FUNCTION_BLOCK FeedOCSLB (* CAT Function Block Type *)
  (* Standard: 61499-2 *)
  (* Version 0.0, 6/7/2026, Schneider Electric, template *)
  PACKAGE SE.Nereda;
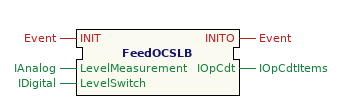
  EVENT_INPUT
    INIT;
  END_EVENT
  EVENT_OUTPUT
    INITO;
  END_EVENT
  SOCKETS
    LevelMeasurement : IAnalog;
    LevelSwitch : IDigital;
  END_SOCKETS
  PLUGS
    IOpCdt : IOpCdtItems;
  END_PLUGS
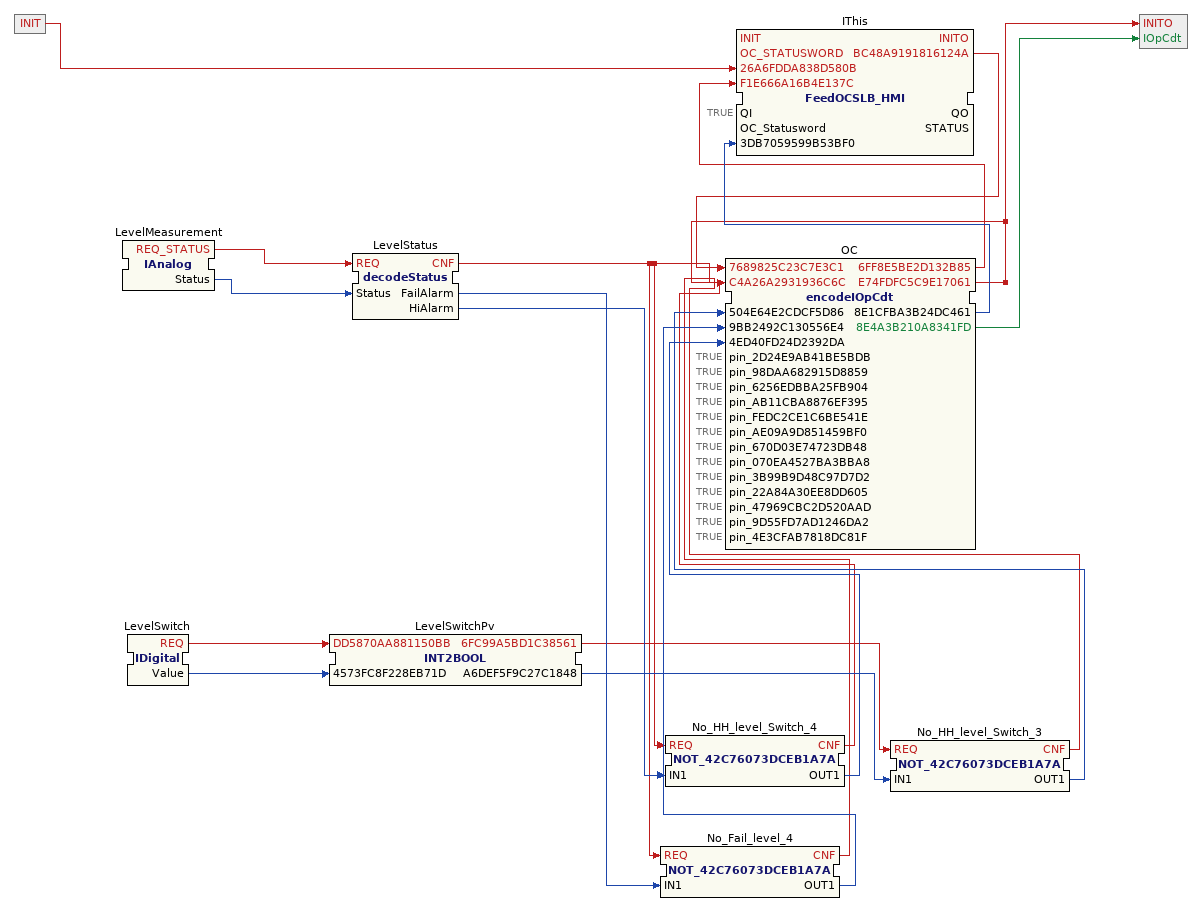
  (* 01 - FUNCTIONNAL INPUT INTERFACE *)
  (* 00 - INITIALIZATION *)
  (* 05 - LOGIC *)
  (* 06 - HMI INTERFACE *)
  (* 03 - FIELD INTERFACE *)
  (* 02 - FUNCTIONNAL OUTPUT INTERFACE *)
  (* Operating Condition Status *)
  (* Operating conditions : 1. Reserved, do not use. 2. No High level in the sludge buffer 49LT0001 3. HighHigh level switch 49LS0002 not activated 4. Level measurement 49LT0001 available *)
  FBS
    OC : encodeIOpCdt(pin_2D24E9AB41BE5BDB := TRUE, pin_98DAA682915D8859 := TRUE, pin_6256EDBBA25FB904 := TRUE, pin_AB11CBA8876EF395 := TRUE, pin_FEDC2CE1C6BE541E := TRUE, pin_AE09A9D851459BF0 := TRUE, pin_670D03E74723DB48 := TRUE, pin_070EA4527BA3BBA8 := TRUE, pin_3B99B9D48C97D7D2 := TRUE, pin_22A84A30EE8DD605 := TRUE, pin_47969CBC2D520AAD := TRUE, pin_9D55FD7AD1246DA2 := TRUE, pin_4E3CFAB7818DC81F := TRUE); (* You set the operating conditions. For the inputs that are not used set a constant to TRUE. *)
    IThis : FeedOCSLB_HMI(QI := TRUE);
    No_HH_level_Switch_3 : NOT_42C76073DCEB1A7A; {SET_ATTRIBUTE(Configuration.GenericFBType.InterfaceParams, Runtime.Standard#CNT:=1;OUT${CNT$}:BOOL)}
    LevelStatus : decodeStatus; {SET_ATTRIBUTE(Configuration.Component.HideUnusedPorts, )}
    LevelSwitchPv : INT2BOOL;
    No_Fail_level_4 : NOT_42C76073DCEB1A7A; {SET_ATTRIBUTE(Configuration.GenericFBType.InterfaceParams, Runtime.Standard#CNT:=1;OUT${CNT$}:BOOL)}
    No_HH_level_Switch_4 : NOT_42C76073DCEB1A7A; {SET_ATTRIBUTE(Configuration.GenericFBType.InterfaceParams, Runtime.Standard#CNT:=1;OUT${CNT$}:BOOL)}
  END_FBS
  EVENT_CONNECTIONS
    INIT TO IThis.26A6FDDA838D580B;
    OC.6FF8E5BE2D132B85 TO IThis.F1E666A16B4E137C;
    IThis.BC48A9191816124A TO OC.7689825C23C7E3C1;
    OC.E74FDFC5C9E17061 TO OC.C4A26A2931936C6C;
    OC.E74FDFC5C9E17061 TO INITO;
    LevelMeasurement.REQ_STATUS TO LevelStatus.REQ;
    LevelSwitch.REQ TO LevelSwitchPv.DD5870AA881150BB;
    LevelSwitchPv.6FC99A5BD1C38561 TO No_HH_level_Switch_3.REQ;
    No_HH_level_Switch_3.CNF TO OC.C4A26A2931936C6C;
    No_Fail_level_4.CNF TO OC.C4A26A2931936C6C;
    LevelStatus.CNF TO OC.C4A26A2931936C6C;
    No_HH_level_Switch_4.CNF TO OC.C4A26A2931936C6C;
    LevelStatus.CNF TO No_HH_level_Switch_4.REQ;
    LevelStatus.CNF TO No_Fail_level_4.REQ;
  END_CONNECTIONS
  DATA_CONNECTIONS
    OC.8E1CFBA3B24DC461 TO IThis.3DB7059599B53BF0;
    LevelMeasurement.Status TO LevelStatus.Status;
    LevelSwitch.Value TO LevelSwitchPv.4573FC8F228EB71D;
    LevelSwitchPv.A6DEF5F9C27C1848 TO No_HH_level_Switch_3.IN1;
    No_HH_level_Switch_3.OUT1 TO OC.504E64E2CDCF5D86;
    LevelStatus.FailAlarm TO No_Fail_level_4.IN1;
    LevelStatus.HiAlarm TO No_HH_level_Switch_4.IN1;
    No_Fail_level_4.OUT1 TO OC.9BB2492C130556E4;
    No_HH_level_Switch_4.OUT1 TO OC.4ED40FD24D2392DA;
  END_CONNECTIONS
  ADAPTER_CONNECTIONS
    OC.8E4A3B210A8341FD TO IOpCdt;
  END_CONNECTIONS
END_FUNCTION_BLOCK
